// TIA Portal project "S7-1500 için Çoklu Girişten İstenileni Seçme(MUX) Komutu" (V18)

(* hardware
DEVICE "S7-1500/ET200MP station_1"  S7-1500 station
   slot 0: "Rail_0"  Rack  6ES7 590-1***0-0AA0
   slot 1: "PLC_1"  CPU 1512C-1 PN  6ES7 512-1CK00-0AB0  V2.8
      slot 3: "CPU display_1"  6ES7591-1AA00-0AA0
      slot 32768: "PROFINET interface_1"  X1
         slot 32769: "Port_1"  X1 P1
         slot 32770: "Port_2"  X1 P2
      slot 34817: "Virtual CP interface port_1"  Virtual CP interface port  Virtual CP interface port
*)

// ===== PLC "PLC_1"  CPU 1512C-1 PN =====

VAR_GLOBAL   // PLC tag table "Default tag table"
   "Tag_1" AT %I0.0 : Bool;
   "Tag_2" AT %MW10 : Int;
   "Tag_3" AT %Q0.0 : Bool;
   "Tag_4" AT %I0.1 : Bool;
   "Tag_5" AT %Q0.1 : Bool;
   "Tag_6" AT %MW11 : Int;
   "Tag_7" AT %MW12 : Int;
   "Tag_8" AT %MW13 : Int;
   "Tag_9" AT %MW14 : Int;
   "Tag_10" AT %I0.2 : Bool;
   "Tag_11" AT %I0.3 : Bool;
END_VAR

// folder: System blocks/Program resources

DATA_BLOCK "IEC_Counter_0_DB"   // DB1
{ S7_Optimized_Access := 'TRUE' }
AUTHOR : Simatic
FAMILY : IEC
NAME : CNTR
VERSION : 1.0
// stored: InstanceOfName IEC_COUNTER
"IEC_COUNTER"
BEGIN
END_DATA_BLOCK

// folder: (top level)

ORGANIZATION_BLOCK "Main"   // OB1, LAD, ProgramCycle
TITLE = "Main Program Sweep (Cycle)"
{ S7_Optimized_Access := 'TRUE' }
VERSION : 0.1
   VAR_INPUT
      Initial_Call : Bool;   // Initial call of this OB
      Remanence : Bool;   // =True, if remanent data are available
   END_VAR
BEGIN

REGION Network 1
   // Sayıcı ile sayma işlemi yapacağız.
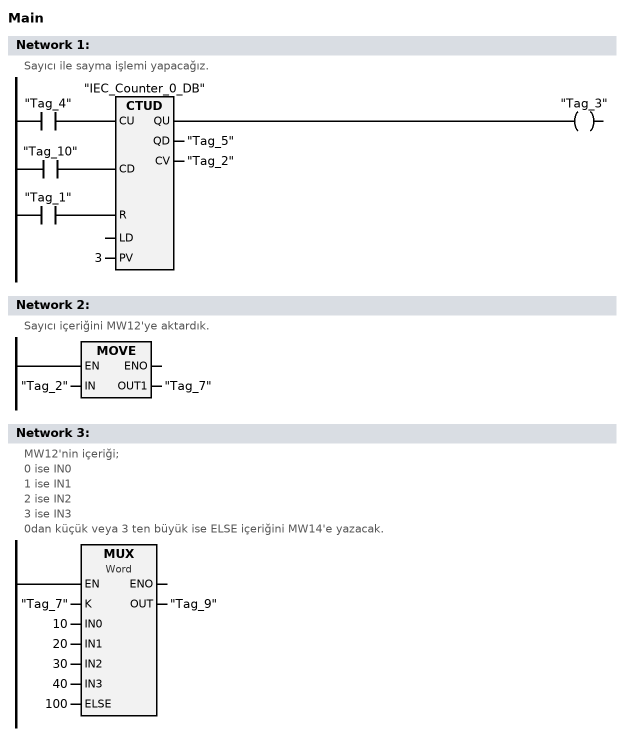
   "IEC_Counter_0_DB".CTUD(CU := "Tag_4", CD := "Tag_10", R := "Tag_1", PV := 3, QD => "Tag_5", CV => "Tag_2");
   "Tag_3" := "IEC_Counter_0_DB".QU;
END_REGION

REGION Network 2
   // Sayıcı içeriğini MW12'ye aktardık.
   RUNG wire#powerrail
      Move(in := "Tag_2", out1 => "Tag_7")
   END_RUNG
   // the same network as SCL:
   "Tag_7" := "Tag_2";
END_REGION

REGION Network 3
   // MW12'nin içeriği;
   // 0 ise IN0
   // 1 ise IN1
   // 2 ise IN2 
   // 3 ise IN3
   // 0dan küçük veya 3 ten büyük ise ELSE içeriğini MW14'e yazacak.
   RUNG wire#powerrail
      { S7_Templates := "SrcType := Word"; S7_GenerateENO := "TRUE" } Mux(k := "Tag_7", in0 := 10, in1 := 20, in2 := 30, in3 := 40, "else" := 100, out => "Tag_9")
   END_RUNG
   // the same network as SCL:
   // no SCL statement known for Mux: written as a call
   Mux(k := "Tag_7", in0 := 10, in1 := 20, in2 := 30, in3 := 40, "else" := 100, out => "Tag_9");
END_REGION
END_ORGANIZATION_BLOCK